(* PLC project Unnamed, Unknown Unnamed 1 *)
(* stored: creationDateTime 2025-03-11T14:10:47, modificationDateTime 2025-03-22T19:23:18 *)

PROGRAM main
  VAR
    St0 : BOOL := 1;
    St1 : BOOL := 0;
    St2 : BOOL := 0;
    StartBut : BOOL := 00;
    BoxBut : BOOL := 0;
    StopBut : BOOL := 0;
    Stepper : BOOL := 0;
    Motor : BOOL := 0;
    STOP : BOOL := 0;
    TON0 : TON;
    TM_DN : BOOL;
  END_VAR
  VAR  (* added by the conversion: wires and edge detectors of the diagram *)
    F_TRIG1 : F_TRIG;
  END_VAR

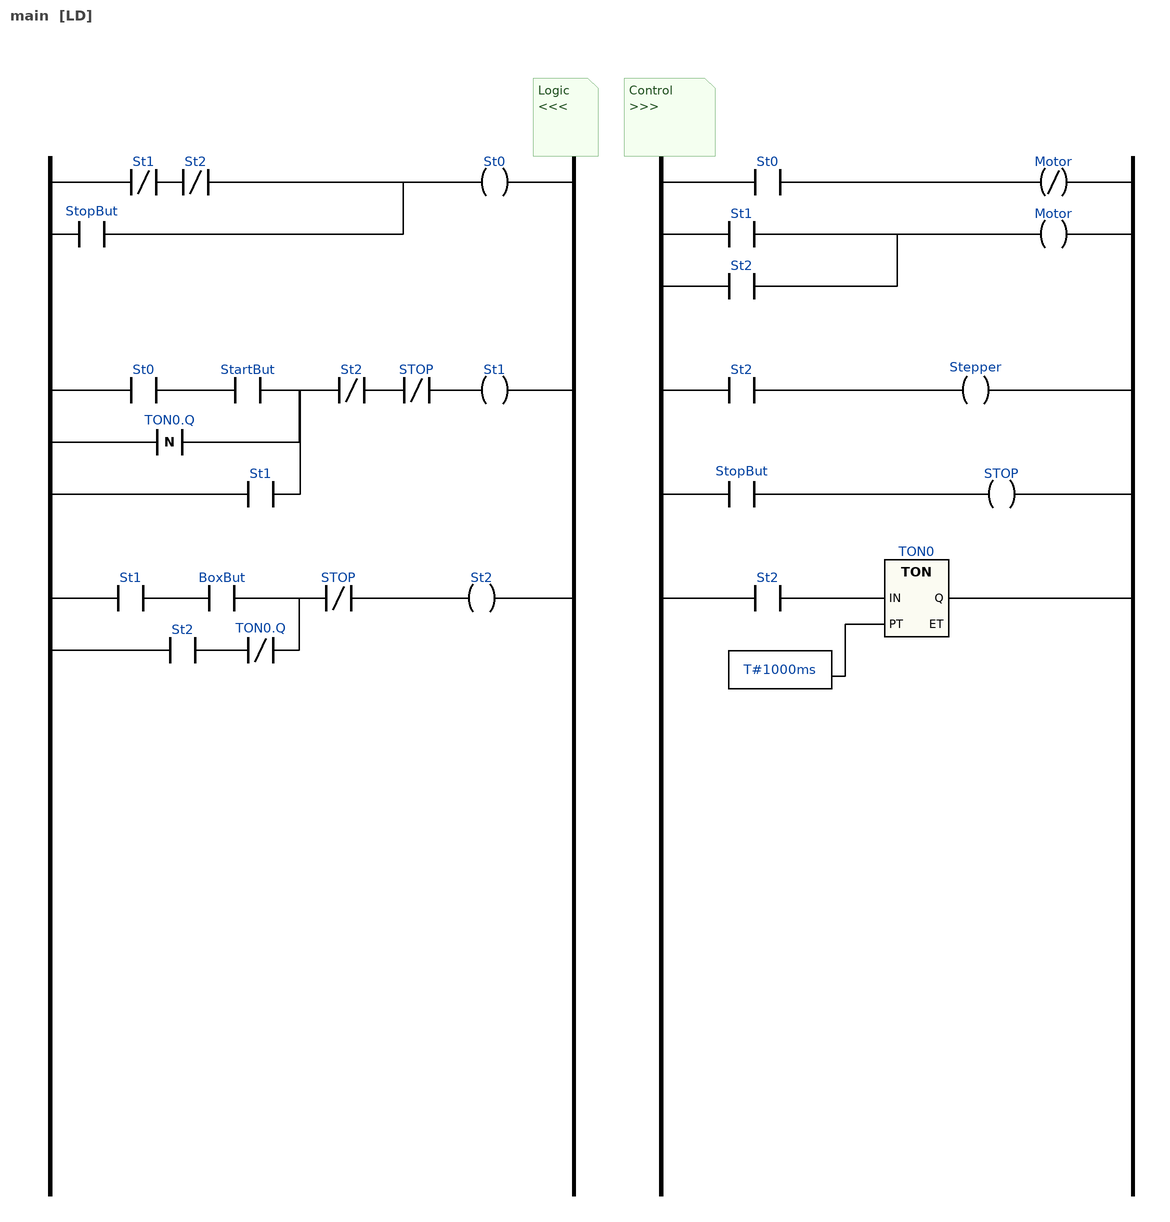
(* LD diagram, written out as Structured Text *)
(* Logic
<<< *)
(* Control
>>> *)
St0 := StopBut OR NOT St1 AND NOT St2;
Motor := NOT St0;
Motor := St1 OR St2;
F_TRIG1(CLK := TON0.Q);
St1 := (St0 AND StartBut OR St1 OR F_TRIG1.Q) AND NOT St2 AND NOT STOP;
St2 := (St1 AND BoxBut OR St2 AND NOT TON0.Q) AND NOT STOP;
Stepper := St2;
STOP := StopBut;
TON0(IN := St2, PT := T#1000ms);
END_PROGRAM

CONFIGURATION Config0
  RESOURCE Res0 ON PLC
    VAR_GLOBAL
      LocalVar0 : DINT;
    END_VAR
    TASK task0(INTERVAL := T#20ms, PRIORITY := 0);
    PROGRAM instance0 WITH task0 : main;
  END_RESOURCE
END_CONFIGURATION
